{attribute 'qualified_only'}
VAR_GLOBAL
	//cycle times
	tTaskCycleTime_MAIN	: TIME := T#50MS;
	tCtrlCycleTime_MAIN	: TIME := T#5S;
	
	//ip addresses
	sIP_EMAG_GT	: STRING := 'opc.tcp://192.168.116.33:4840';
END_VAR

(* stored: Version 1.1.0.1, ProductVersion 3.1.4024.10
   GVL GlobalVariables: Id {03b0febb-bd51-42dd-a1dc-b1b77f4022cb} *)
